{attribute 'qualified_only'}
{attribute 'strict'}
TYPE LEDColor :
(
	Off,
	Red,
	Green,
	Blue
);
END_TYPE

(* stored: Version 1.1.0.1, ProductVersion 3.1.4024.12
   DUT LEDColor: Id {c987c291-d13f-4bdb-aff4-8a7d8b4aadca} *)
